FUNCTION_BLOCK PuestoAutomatico
VAR_INPUT
	Reset:BOOL;
	SFCreset:BOOL;
	Enable:BOOL;
	FinCiclo:BOOL;
	SensorPallet:BOOL;
	Pulsador1 AT %I*:BOOL;

	NumeroDePuesto :INT;
	
	SelectorByPass AT %I*:BOOL;
	Pass AT %I*:BOOL;
	Fail AT %I*:BOOL;
	
	SensorPieza1 AT %I*:BOOL;
	SensorPieza2 AT %I*:BOOL;
	
END_VAR
VAR_OUTPUT
	
	Ready AT %Q*:BOOL;
	StopperOFF AT %Q*:BOOL;
	Centrador AT%Q*:BOOL;
	LuzAmbar AT%Q*:BOOL;
	SalidaAlarma:BOOL;
	EnMovimiento:BOOL;
	EsperandoPalet:BOOL;
	RetrasoPuesto :INT;
	FinPuesto:BOOL;
	
	
	
END_VAR
VAR
END_VAR

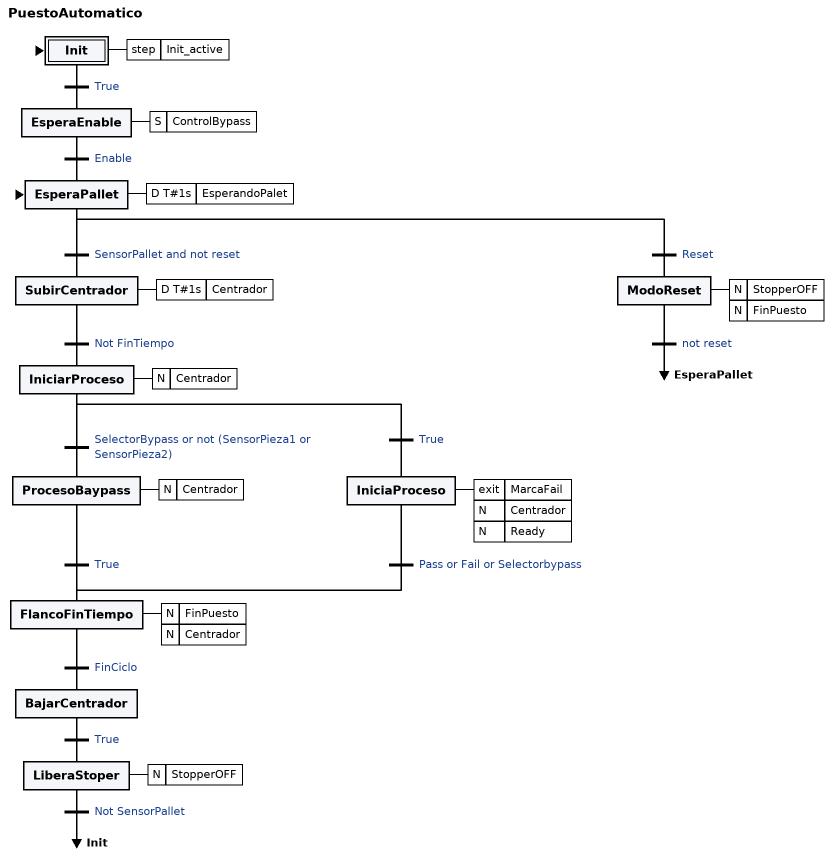
INITIAL_STEP Init:
    Init_active(N);  // step action
END_STEP
TRANSITION FROM Init TO EsperaEnable
    := True;
END_TRANSITION
STEP EsperaEnable:
    ControlBypass(S);
END_STEP
TRANSITION FROM EsperaEnable TO EsperaPallet
    := Enable;
END_TRANSITION
STEP EsperaPallet:
    EsperandoPalet(D, T#1s);
END_STEP
TRANSITION FROM EsperaPallet TO SubirCentrador
    := SensorPallet and not reset;
END_TRANSITION
STEP SubirCentrador:  // min time T#2s
    Centrador(D, T#1s);
END_STEP
TRANSITION FROM SubirCentrador TO IniciarProceso
    := Not FinTiempo;
END_TRANSITION
STEP IniciarProceso:
    Centrador(N);
END_STEP
TRANSITION FROM IniciarProceso TO ProcesoBaypass
    := SelectorBypass or not (SensorPieza1 or SensorPieza2);
END_TRANSITION
STEP ProcesoBaypass:
    Centrador(N);
END_STEP
TRANSITION FROM ProcesoBaypass TO FlancoFinTiempo
    := True;
END_TRANSITION
TRANSITION FROM IniciarProceso TO IniciaProceso
    := True;
END_TRANSITION
STEP IniciaProceso:
    MarcaFail(P0);  // exit action
    Centrador(N);
    Ready(N);
END_STEP
TRANSITION FROM IniciaProceso TO FlancoFinTiempo
    := Pass or Fail or Selectorbypass;
END_TRANSITION
STEP FlancoFinTiempo:
    FinPuesto(N);
    Centrador(N);
END_STEP
TRANSITION FROM FlancoFinTiempo TO BajarCentrador
    := FinCiclo;
END_TRANSITION
STEP BajarCentrador:  // min time T#1s
END_STEP
TRANSITION FROM BajarCentrador TO LiberaStoper
    := True;
END_TRANSITION
TRANSITION FROM EsperaPallet TO ModoReset
    := Reset;
END_TRANSITION
STEP ModoReset:
    StopperOFF(N);
    FinPuesto(N);
END_STEP
TRANSITION FROM ModoReset TO EsperaPallet
    := not reset;
END_TRANSITION
STEP LiberaStoper:  // min time T#1s
    StopperOFF(N);
END_STEP
TRANSITION FROM LiberaStoper TO Init
    := Not SensorPallet;
END_TRANSITION

ACTION ControlBypass:
LuzAmbar := SelectorByPass;
END_ACTION

ACTION Init_active:
FinPUesto :=FALSE;
SFCreset:=FALSE;
END_ACTION

ACTION MarcaFail:
IF  Fail = TRUE THEN 
	gvl.FalloPallet[NumeroDePuesto] := TRUE;
END_IF
END_ACTION

END_FUNCTION_BLOCK

(* stored: Version 1.1.0.1, ProductVersion 3.1.4024.3
   POU PuestoAutomatico: Id {6ab4d035-a3b6-4dbd-a585-9d93cc4d0d81}, SpecialFunc None
   Action ControlBypass: Id {89abec94-fd16-499d-aeb0-e0d06e2e59cd}
   Action Init_active: Id {dde9dbee-2ac5-460e-b73a-8cc9db847f61}
   Action MarcaFail: Id {60a22124-027a-4780-8ffe-50eb5b2dc2be} *)
